FUNCTION_BLOCK plant (* ODE *)
  (* Standard: 61499-2 *)
  (* Version 0.1, 2017-00-25, hpea485, UOA *)
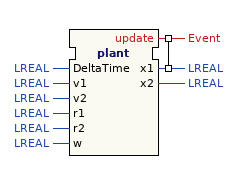
  EVENT_OUTPUT
    update WITH x0, x1;
  END_EVENT
  VAR_INPUT
    DeltaTime : LREAL := 0.01;
    v1 : LREAL := 0.5;
    v2 : LREAL := 0.5;
    r1 : LREAL := 0.25;
    r2 : LREAL := 0.25;
    w : LREAL := 1;
  END_VAR
  VAR_OUTPUT
    x1 : LREAL;
    x2 : LREAL;
  END_VAR
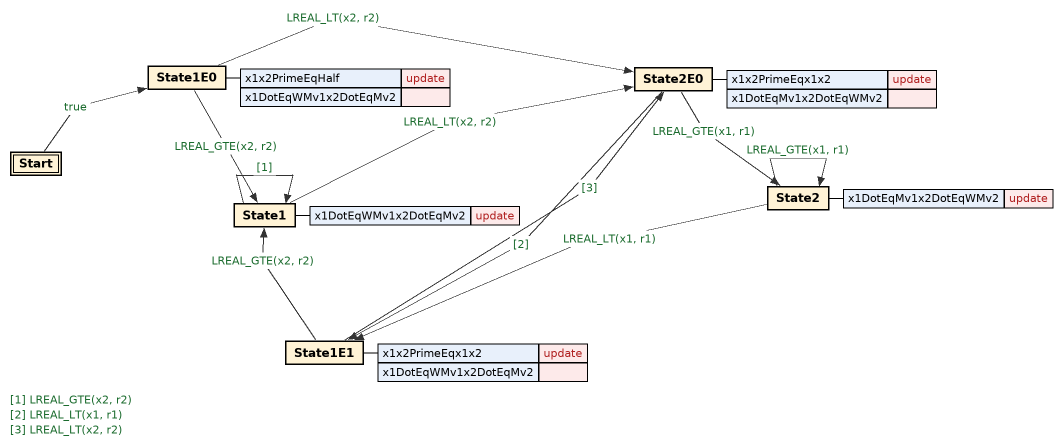
  EC_STATES
    Start;
    State1E0 : x1x2PrimeEqHalf -> update, x1DotEqWMv1x2DotEqMv2;
    State1 : x1DotEqWMv1x2DotEqMv2 -> update;
    State2E0 : x1x2PrimeEqx1x2 -> update, x1DotEqMv1x2DotEqWMv2;
    State2 : x1DotEqMv1x2DotEqWMv2 -> update;
    State1E1 : x1x2PrimeEqx1x2 -> update, x1DotEqWMv1x2DotEqMv2;
  END_STATES
  EC_TRANSITIONS
    Start TO State1E0 := true;
    State1E0 TO State2E0 := LREAL_LT(x2, r2);
    State1E0 TO State1 := LREAL_GTE(x2, r2);
    State1 TO State2E0 := LREAL_LT(x2, r2);
    State1 TO State1 := LREAL_GTE(x2, r2);
    State2E0 TO State1E1 := LREAL_LT(x1, r1);
    State2E0 TO State2 := LREAL_GTE(x1, r1);
    State2 TO State1E1 := LREAL_LT(x1, r1);
    State2 TO State2 := LREAL_GTE(x1, r1);
    State1E1 TO State2E0 := LREAL_LT(x2, r2);
    State1E1 TO State1 := LREAL_GTE(x2, r2);
  END_TRANSITIONS
  ALGORITHM x1x2PrimeEqHalf IN C: (* ODE_init *)
x1_prime = 0.5;
x2_prime = 0.5;
  END_ALGORITHM
  ALGORITHM x1x2PrimeEqx1x2 IN C: (* ODE_init *)
x1_prime = x1;
x2_prime = x2;
  END_ALGORITHM
  ALGORITHM x1DotEqWMv1x2DotEqMv2 IN C: (* ODE *)
x1_dot = w - v1;
x2_dot = -v2;
  END_ALGORITHM
  ALGORITHM x1DotEqMv1x2DotEqWMv2 IN C: (* ODE *)
x1_dot = -v1;
x2_dot = w - v2;
  END_ALGORITHM
END_FUNCTION_BLOCK
